KUKA KRL data list: Up777.dat

&ACCESS RVP
&REL 11
&PARAM EDITMASK = Up999[1-999]
&PARAM TPVW_VERSION = 8.3.17
&PARAM TEMPLATE = C:\KRC\Roboter\Template\upvorgabe
DEFDAT UP777
; FOLD ;%{H} %MKUKATPVW
; ENDFOLD
; interface to basic routines
 EXT  BAS (BAS_COMMAND  :IN,REAL  :IN )
; interface to VW-standard routines
EXT VW (VW_COMMAND:IN, BOOL: IN, REAL:IN, REAL:IN, REAL:IN, REAL:IN, BOOL :IN, E6POS :IN )
; interface to VW_USER - Call
EXT  VW_USER (VW_USER_CMD :IN,INT :IN,REAL  :IN,REAL  :IN,REAL  :IN,REAL  :IN,REAL  :IN,REAL  :IN,REAL  :IN,REAL  :IN,REAL  :IN,BOOL  :IN)
EXT  VW_USR_R (VW_USER_CMD :IN,INT :IN,REAL  :IN,REAL  :IN,REAL  :IN,REAL  :IN,REAL  :IN,REAL  :IN,REAL  :IN,REAL  :IN,REAL  :IN,BOOL  :IN)
EXT  IBGN (IBGN_COMMAND  :IN,BOOL  :IN,REAL  :IN,REAL  :IN,BOOL  :IN,E6POS  :OUT )
; interface select routine
EXTFCT INT  SELECT (SUBTYPE  :IN,INT  :IN,BOOL  :IN,ARI_TYP  :IN,INT  :IN,BOOL_TYP  :IN,INT  :IN,BOOL  :IN)
INT VW_NEXT_FREE = 3
INT VW_NFREE_SPS = 3
INT VW_MAX_SPS = 103
DECL VW_MPARA_TYP P1_D = {TOOL_NO 3,BASE_NO 0,VB 100,VE 0,ACC 100,TRG_TIME 0,MOVE_TYPE #PTP_MOTION}
DECL E6POS P1 = {X 296.8807, Y 1596.921, Z 1022.207, A 135.347, B 84.03362, C 81.37661, S 2, T 3 , E1 -518.8434, E2 0.0, E3 0.0, E4 0.0, E5 0.0, E6 0.0}
DECL VW_MPARA_TYP P2_D = {TOOL_NO 3,BASE_NO 0,VB 100,VE 0,ACC 100,TRG_TIME 0,MOVE_TYPE #PTP_MOTION}
DECL E6POS P2 = {X 296.8807, Y 1596.921, Z 1022.207, A 135.347, B 84.03362, C 81.37661, S 2, T 3 , E1 -518.8434, E2 0.0, E3 0.0, E4 0.0, E5 0.0, E6 0.0}
ENDDAT
